// TIA Portal V20 export
DATA_BLOCK "Config"   // DB45
{ DB_Accessible_From_OPC_UA := 'FALSE' }
AUTHOR : ERsystem_FA2_DH. Kim
// stored: Access Published, DBAccessibleFromOPCUA false, DBAccessibleFromWebserver false, MemoryReserve 100, Namespace Unit1.Em7
   VAR RETAIN
      em { ExternalAccessible := 'False'; ExternalVisible := 'False'; ExternalWritable := 'False'} : "LAF_typeEmConfiguration";
      axis { ExternalAccessible := 'False'; ExternalVisible := 'False'; ExternalWritable := 'False'} : Array[1.._.U1EM7_NO_OF_AXES] of DB_ANY;
      cam { ExternalAccessible := 'False'; ExternalVisible := 'False'; ExternalWritable := 'False'} : Array[1.._.U1EM7_NO_OF_CAM] of DB_ANY;
      cmSepaClampDetectSensor { ExternalAccessible := 'False'; ExternalVisible := 'False'; ExternalWritable := 'False'} : "LBC_typeDigitalSignalConfiguration";
      cmSepaGripperDetectSensor { ExternalAccessible := 'False'; ExternalVisible := 'False'; ExternalWritable := 'False'} : "LBC_typeDigitalSignalConfiguration";
      cmJRWinderDetectSensor { ExternalAccessible := 'False'; ExternalVisible := 'False'; ExternalWritable := 'False'} : "LBC_typeDigitalSignalConfiguration";
      cmSepaClampSafetyPinDetectSensor { ExternalAccessible := 'False'; ExternalVisible := 'False'; ExternalWritable := 'False'} : "LBC_typeDigitalSignalConfiguration";
      cmSepaGripperSafetyPinDetectSensor { ExternalAccessible := 'False'; ExternalVisible := 'False'; ExternalWritable := 'False'} : "LBC_typeDigitalSignalConfiguration";
      cmSepaClampnCutterAxisX { ExternalAccessible := 'False'; ExternalVisible := 'False'; ExternalWritable := 'False'} : "LBC_typeAxis64PosConfiguration";
      cmSepaClampnCutterAxisZ { ExternalAccessible := 'False'; ExternalVisible := 'False'; ExternalWritable := 'False'} : "LBC_typeAxis64PosConfiguration";
      cmSepaGripperAxisX { ExternalAccessible := 'False'; ExternalVisible := 'False'; ExternalWritable := 'False'} : "LBC_typeAxis64PosConfiguration";
      cmSepaGripperAxisZ { ExternalAccessible := 'False'; ExternalVisible := 'False'; ExternalWritable := 'False'} : "LBC_typeAxis64PosConfiguration";
      cmSepaGripperAxisC { ExternalAccessible := 'False'; ExternalVisible := 'False'; ExternalWritable := 'False'} : "LBC_typeAxis64PosConfiguration";
      cmJRWinderRearAxisY { ExternalAccessible := 'False'; ExternalVisible := 'False'; ExternalWritable := 'False'} : "LBC_typeAxis64PosConfiguration";
      cmJRWinderFrontAxisY { ExternalAccessible := 'False'; ExternalVisible := 'False'; ExternalWritable := 'False'} : "LBC_typeAxis64PosConfiguration";
      cmJRWinderAxisB { ExternalAccessible := 'False'; ExternalVisible := 'False'; ExternalWritable := 'False'} : "LBC_typeAxis64PosConfiguration";
      cmJRPusherAxisZ { ExternalAccessible := 'False'; ExternalVisible := 'False'; ExternalWritable := 'False'} : "LBC_typeAxis64PosConfiguration";
      cmSepaCutterUpDown { ExternalAccessible := 'False'; ExternalVisible := 'False'; ExternalWritable := 'False'} : "LBC_typeTwoWayActuatorConfiguration";
      cmSepaClampTopUpDown { ExternalAccessible := 'False'; ExternalVisible := 'False'; ExternalWritable := 'False'} : "LBC_typeTwoWayActuatorConfiguration";
      cmSepaClampBottomUpDown { ExternalAccessible := 'False'; ExternalVisible := 'False'; ExternalWritable := 'False'} : "LBC_typeTwoWayActuatorConfiguration";
      cmStackGripperOpenClose { ExternalAccessible := 'False'; ExternalVisible := 'False'; ExternalWritable := 'False'} : "LBC_typeTwoWayActuatorConfiguration";
      cmStackGripperFwdBwd { ExternalAccessible := 'False'; ExternalVisible := 'False'; ExternalWritable := 'False'} : "LBC_typeTwoWayActuatorConfiguration";
      cmJRWinderClampTopRearUpDown { ExternalAccessible := 'False'; ExternalVisible := 'False'; ExternalWritable := 'False'} : "LBC_typeTwoWayActuatorConfiguration";
      cmJRWinderClampBtmRearUpDown { ExternalAccessible := 'False'; ExternalVisible := 'False'; ExternalWritable := 'False'} : "LBC_typeTwoWayActuatorConfiguration";
      cmJRWinderClampTopFrontUpDown { ExternalAccessible := 'False'; ExternalVisible := 'False'; ExternalWritable := 'False'} : "LBC_typeTwoWayActuatorConfiguration";
      cmJRWinderClampBtmFrontUpDown { ExternalAccessible := 'False'; ExternalVisible := 'False'; ExternalWritable := 'False'} : "LBC_typeTwoWayActuatorConfiguration";
      cmPusherRollerUpDown { ExternalAccessible := 'False'; ExternalVisible := 'False'; ExternalWritable := 'False'} : "LBC_typeTwoWayActuatorConfiguration";
      cmPusherRollerFwdBwd { ExternalAccessible := 'False'; ExternalVisible := 'False'; ExternalWritable := 'False'} : "LBC_typeTwoWayActuatorConfiguration";
      softCam : Struct
         cmSepaClampnCutterAxisX : "LER_typeSoftCamInterface";
         cmSepaClampnCutterAxisZ { S7_SetPoint := 'True'} : "LER_typeSoftCamInterface";
         cmSepaGripperAxisX { S7_SetPoint := 'True'} : "LER_typeSoftCamInterface";
         cmSepaGripperAxisZ { S7_SetPoint := 'True'} : "LER_typeSoftCamInterface";
         cmSepaGripperAxisC { S7_SetPoint := 'True'} : "LER_typeSoftCamInterface";
         cmJRWinderRearAxisY { S7_SetPoint := 'True'} : "LER_typeSoftCamInterface";
         cmJRWinderFrontAxisY { S7_SetPoint := 'True'} : "LER_typeSoftCamInterface";
         cmJRWinderAxisB { S7_SetPoint := 'True'} : "LER_typeSoftCamInterface";
         cmJRPusherAxisZ { S7_SetPoint := 'True'} : "LER_typeSoftCamInterface";
      END_STRUCT;
   END_VAR
BEGIN
   em.referenceDesignator.parent := WSTRING#'';
   em.referenceDesignator.relative := WSTRING#'';
   em.referenceDesignator.combined := WSTRING#'';
   axis[1] := 177;   // SepaClampnCutterAxisX
   axis[2] := 175;   // SepaClampnCutterAxisZ
   axis[3] := 178;   // SepaGripperAxisX
   axis[4] := 173;   // SepaGripperAxisZ
   axis[5] := 174;   // SepaGripperAxisC
   axis[6] := 180;   // JRWinderRearAxisY
   axis[7] := 179;   // JRWinderFrontAxisY
   axis[8] := 176;   // JRWinderAxisB
   axis[9] := 141;   // JRPusherAxisZ
   cam[1] := 184;
   cam[2] := 23;
   cam[3] := 266;
   cam[4] := 47;
   cam[5] := 390;
   cam[6] := 80;
   cmSepaClampDetectSensor.referenceDesignator := WSTRING#'DigitalSignal';
   cmSepaClampDetectSensor.onDelay := T#0MS;
   cmSepaClampDetectSensor.offDelay := T#0MS;
   cmSepaClampDetectSensor.default := FALSE;
   cmSepaClampDetectSensor.invertProcessValue := FALSE;
   cmSepaClampDetectSensor.disableAlarms := FALSE;
   cmSepaGripperDetectSensor.referenceDesignator := WSTRING#'DigitalSignal';
   cmSepaGripperDetectSensor.onDelay := T#0MS;
   cmSepaGripperDetectSensor.offDelay := T#0MS;
   cmSepaGripperDetectSensor.default := FALSE;
   cmSepaGripperDetectSensor.invertProcessValue := FALSE;
   cmSepaGripperDetectSensor.disableAlarms := FALSE;
   cmJRWinderDetectSensor.referenceDesignator := WSTRING#'DigitalSignal';
   cmJRWinderDetectSensor.onDelay := T#0MS;
   cmJRWinderDetectSensor.offDelay := T#0MS;
   cmJRWinderDetectSensor.default := FALSE;
   cmJRWinderDetectSensor.invertProcessValue := FALSE;
   cmJRWinderDetectSensor.disableAlarms := FALSE;
   cmSepaClampSafetyPinDetectSensor.referenceDesignator := WSTRING#'DigitalSignal';
   cmSepaClampSafetyPinDetectSensor.onDelay := T#0MS;
   cmSepaClampSafetyPinDetectSensor.offDelay := T#0MS;
   cmSepaClampSafetyPinDetectSensor.default := FALSE;
   cmSepaClampSafetyPinDetectSensor.invertProcessValue := FALSE;
   cmSepaClampSafetyPinDetectSensor.disableAlarms := FALSE;
   cmSepaGripperSafetyPinDetectSensor.referenceDesignator := WSTRING#'DigitalSignal';
   cmSepaGripperSafetyPinDetectSensor.onDelay := T#0MS;
   cmSepaGripperSafetyPinDetectSensor.offDelay := T#0MS;
   cmSepaGripperSafetyPinDetectSensor.default := FALSE;
   cmSepaGripperSafetyPinDetectSensor.invertProcessValue := FALSE;
   cmSepaGripperSafetyPinDetectSensor.disableAlarms := FALSE;
   cmSepaClampnCutterAxisX.referenceDesignator := WSTRING#'SepaClampnCutterAxisX';
   cmSepaClampnCutterAxisX.disableAlarms := FALSE;
   cmSepaClampnCutterAxisX.masterControlPopUp := TRUE;
   cmSepaClampnCutterAxisX.setPositions[0].position := 100.0;
   cmSepaClampnCutterAxisX.setPositions[1].position := 0.0;
   cmSepaClampnCutterAxisX.setPositions[2].position := 200.0;
   cmSepaClampnCutterAxisX.setPositions[3].position := 106.125;
   cmSepaClampnCutterAxisX.setPositions[4].position := 212.25;
   cmSepaClampnCutterAxisX.setPositions[5].position := 318.375;
   cmSepaClampnCutterAxisX.setPositions[6].position := 424.5;
   cmSepaClampnCutterAxisX.setPositions[7].position := 600.0;
   cmSepaClampnCutterAxisX.setPositions[8..15].position := 0.0;
   cmSepaClampnCutterAxisX.setPositions[0..2].velocity := 100.0;
   cmSepaClampnCutterAxisX.setPositions[3..6].velocity := -1.17916666666667;
   cmSepaClampnCutterAxisX.setPositions[7].velocity := 100.0;
   cmSepaClampnCutterAxisX.setPositions[8..15].velocity := -1.0;
   cmSepaClampnCutterAxisX.setPositions[0..2].acceleration := 1000.0;
   cmSepaClampnCutterAxisX.setPositions[3..6].acceleration := -11.7916666666667;
   cmSepaClampnCutterAxisX.setPositions[7].acceleration := 1000.0;
   cmSepaClampnCutterAxisX.setPositions[8..15].acceleration := -1.0;
   cmSepaClampnCutterAxisX.setPositions[0..2].deceleration := 1000.0;
   cmSepaClampnCutterAxisX.setPositions[3..6].deceleration := -11.7916666666667;
   cmSepaClampnCutterAxisX.setPositions[7].deceleration := 1000.0;
   cmSepaClampnCutterAxisX.setPositions[8..15].deceleration := -1.0;
   cmSepaClampnCutterAxisX.setPositions[0..15]."name" := '';
   cmSepaClampnCutterAxisZ.referenceDesignator := WSTRING#'SepaClampnCutterAxisZ';
   cmSepaClampnCutterAxisZ.disableAlarms := FALSE;
   cmSepaClampnCutterAxisZ.masterControlPopUp := TRUE;
   cmSepaClampnCutterAxisZ.setPositions[0].position := 0.0;
   cmSepaClampnCutterAxisZ.setPositions[1].position := 25.0;
   cmSepaClampnCutterAxisZ.setPositions[2].position := 50.0;
   cmSepaClampnCutterAxisZ.setPositions[3].position := -106.125;
   cmSepaClampnCutterAxisZ.setPositions[4..15].position := 0.0;
   cmSepaClampnCutterAxisZ.setPositions[0..2].velocity := 50.0;
   cmSepaClampnCutterAxisZ.setPositions[3..4].velocity := -1.17916666666667;
   cmSepaClampnCutterAxisZ.setPositions[5..15].velocity := -1.0;
   cmSepaClampnCutterAxisZ.setPositions[0..2].acceleration := 500.0;
   cmSepaClampnCutterAxisZ.setPositions[3..4].acceleration := -11.7916666666667;
   cmSepaClampnCutterAxisZ.setPositions[5..15].acceleration := -1.0;
   cmSepaClampnCutterAxisZ.setPositions[0..2].deceleration := 500.0;
   cmSepaClampnCutterAxisZ.setPositions[3..4].deceleration := -11.7916666666667;
   cmSepaClampnCutterAxisZ.setPositions[5..15].deceleration := -1.0;
   cmSepaClampnCutterAxisZ.setPositions[0..15]."name" := '';
   cmSepaGripperAxisX.referenceDesignator := WSTRING#'SepaGripperAxisX';
   cmSepaGripperAxisX.disableAlarms := FALSE;
   cmSepaGripperAxisX.masterControlPopUp := TRUE;
   cmSepaGripperAxisX.setPositions[0].position := 100.0;
   cmSepaGripperAxisX.setPositions[1].position := 400.0;
   cmSepaGripperAxisX.setPositions[2].position := 300.0;
   cmSepaGripperAxisX.setPositions[3].position := 150.0;
   cmSepaGripperAxisX.setPositions[4].position := 250.0;
   cmSepaGripperAxisX.setPositions[5].position := 100.0;
   cmSepaGripperAxisX.setPositions[6..15].position := 0.0;
   cmSepaGripperAxisX.setPositions[0..6].velocity := 100.0;
   cmSepaGripperAxisX.setPositions[7..15].velocity := -1.0;
   cmSepaGripperAxisX.setPositions[0..6].acceleration := 1000.0;
   cmSepaGripperAxisX.setPositions[7..15].acceleration := -1.0;
   cmSepaGripperAxisX.setPositions[0..6].deceleration := 1000.0;
   cmSepaGripperAxisX.setPositions[7..15].deceleration := -1.0;
   cmSepaGripperAxisX.setPositions[0..15]."name" := '';
   cmSepaGripperAxisZ.referenceDesignator := WSTRING#'SepaGripperAxisZ';
   cmSepaGripperAxisZ.disableAlarms := FALSE;
   cmSepaGripperAxisZ.masterControlPopUp := TRUE;
   cmSepaGripperAxisZ.setPositions[0].position := 0.0;
   cmSepaGripperAxisZ.setPositions[1].position := 25.0;
   cmSepaGripperAxisZ.setPositions[2].position := 2.0;
   cmSepaGripperAxisZ.setPositions[3].position := 3.0;
   cmSepaGripperAxisZ.setPositions[4].position := 4.0;
   cmSepaGripperAxisZ.setPositions[5].position := 5.0;
   cmSepaGripperAxisZ.setPositions[6].position := 50.0;
   cmSepaGripperAxisZ.setPositions[7..15].position := 0.0;
   cmSepaGripperAxisZ.setPositions[0..6].velocity := 50.0;
   cmSepaGripperAxisZ.setPositions[7..15].velocity := -1.0;
   cmSepaGripperAxisZ.setPositions[0..6].acceleration := 500.0;
   cmSepaGripperAxisZ.setPositions[7..15].acceleration := -1.0;
   cmSepaGripperAxisZ.setPositions[0..6].deceleration := 500.0;
   cmSepaGripperAxisZ.setPositions[7..15].deceleration := -1.0;
   cmSepaGripperAxisZ.setPositions[0..15]."name" := '';
   cmSepaGripperAxisC.referenceDesignator := WSTRING#'SepaGripperAxisC';
   cmSepaGripperAxisC.disableAlarms := FALSE;
   cmSepaGripperAxisC.masterControlPopUp := TRUE;
   cmSepaGripperAxisC.setPositions[0].position := 0.0;
   cmSepaGripperAxisC.setPositions[1].position := 180.0;
   cmSepaGripperAxisC.setPositions[2].position := 90.0;
   cmSepaGripperAxisC.setPositions[3..15].position := 0.0;
   cmSepaGripperAxisC.setPositions[0..2].velocity := 100.0;
   cmSepaGripperAxisC.setPositions[3..15].velocity := -1.0;
   cmSepaGripperAxisC.setPositions[0..2].acceleration := 1000.0;
   cmSepaGripperAxisC.setPositions[3..15].acceleration := -1.0;
   cmSepaGripperAxisC.setPositions[0..2].deceleration := 1000.0;
   cmSepaGripperAxisC.setPositions[3..15].deceleration := -1.0;
   cmSepaGripperAxisC.setPositions[0..15]."name" := '';
   cmJRWinderRearAxisY.referenceDesignator := WSTRING#'JRWinderRearAxisY';
   cmJRWinderRearAxisY.disableAlarms := FALSE;
   cmJRWinderRearAxisY.masterControlPopUp := TRUE;
   cmJRWinderRearAxisY.setPositions[0].position := 0.0;
   cmJRWinderRearAxisY.setPositions[1].position := 50.0;
   cmJRWinderRearAxisY.setPositions[2..15].position := 0.0;
   cmJRWinderRearAxisY.setPositions[0..1].velocity := 50.0;
   cmJRWinderRearAxisY.setPositions[2..15].velocity := -1.0;
   cmJRWinderRearAxisY.setPositions[0..1].acceleration := 500.0;
   cmJRWinderRearAxisY.setPositions[2..15].acceleration := -1.0;
   cmJRWinderRearAxisY.setPositions[0..1].deceleration := 500.0;
   cmJRWinderRearAxisY.setPositions[2..15].deceleration := -1.0;
   cmJRWinderRearAxisY.setPositions[0..15]."name" := '';
   cmJRWinderFrontAxisY.referenceDesignator := WSTRING#'JRWinderFrontAxisY';
   cmJRWinderFrontAxisY.disableAlarms := FALSE;
   cmJRWinderFrontAxisY.masterControlPopUp := TRUE;
   cmJRWinderFrontAxisY.setPositions[0].position := 0.0;
   cmJRWinderFrontAxisY.setPositions[1].position := 50.0;
   cmJRWinderFrontAxisY.setPositions[2..15].position := 0.0;
   cmJRWinderFrontAxisY.setPositions[0..1].velocity := 50.0;
   cmJRWinderFrontAxisY.setPositions[2..15].velocity := -1.0;
   cmJRWinderFrontAxisY.setPositions[0..1].acceleration := 500.0;
   cmJRWinderFrontAxisY.setPositions[2..15].acceleration := -1.0;
   cmJRWinderFrontAxisY.setPositions[0..1].deceleration := 500.0;
   cmJRWinderFrontAxisY.setPositions[2..15].deceleration := -1.0;
   cmJRWinderFrontAxisY.setPositions[0..15]."name" := '';
   cmJRWinderAxisB.referenceDesignator := WSTRING#'JRWinderAxisB';
   cmJRWinderAxisB.disableAlarms := FALSE;
   cmJRWinderAxisB.masterControlPopUp := TRUE;
   cmJRWinderAxisB.setPositions[0].position := 0.0;
   cmJRWinderAxisB.setPositions[1].position := 90.0;
   cmJRWinderAxisB.setPositions[2].position := 180.0;
   cmJRWinderAxisB.setPositions[3].position := 270.0;
   cmJRWinderAxisB.setPositions[4].position := 360.0;
   cmJRWinderAxisB.setPositions[5].position := 450.0;
   cmJRWinderAxisB.setPositions[6].position := 540.0;
   cmJRWinderAxisB.setPositions[7].position := 360.0;
   cmJRWinderAxisB.setPositions[8].position := 540.0;
   cmJRWinderAxisB.setPositions[9..15].position := 0.0;
   cmJRWinderAxisB.setPositions[0..8].velocity := 100.0;
   cmJRWinderAxisB.setPositions[9..15].velocity := -1.0;
   cmJRWinderAxisB.setPositions[0..8].acceleration := 1000.0;
   cmJRWinderAxisB.setPositions[9..15].acceleration := -1.0;
   cmJRWinderAxisB.setPositions[0..8].deceleration := 1000.0;
   cmJRWinderAxisB.setPositions[9..15].deceleration := -1.0;
   cmJRWinderAxisB.setPositions[0..15]."name" := '';
   cmJRPusherAxisZ.referenceDesignator := WSTRING#'JRPusherAxisZ';
   cmJRPusherAxisZ.disableAlarms := FALSE;
   cmJRPusherAxisZ.masterControlPopUp := TRUE;
   cmJRPusherAxisZ.setPositions[0].position := 0.0;
   cmJRPusherAxisZ.setPositions[1].position := 100.0;
   cmJRPusherAxisZ.setPositions[2].position := -106.125;
   cmJRPusherAxisZ.setPositions[3..15].position := 0.0;
   cmJRPusherAxisZ.setPositions[0..1].velocity := 100.0;
   cmJRPusherAxisZ.setPositions[2..3].velocity := -1.17916666666667;
   cmJRPusherAxisZ.setPositions[4..15].velocity := -1.0;
   cmJRPusherAxisZ.setPositions[0..1].acceleration := 1000.0;
   cmJRPusherAxisZ.setPositions[2..3].acceleration := -11.7916666666667;
   cmJRPusherAxisZ.setPositions[4..15].acceleration := -1.0;
   cmJRPusherAxisZ.setPositions[0..1].deceleration := 1000.0;
   cmJRPusherAxisZ.setPositions[2..3].deceleration := -11.7916666666667;
   cmJRPusherAxisZ.setPositions[4..15].deceleration := -1.0;
   cmJRPusherAxisZ.setPositions[0..15]."name" := '';
   cmSepaCutterUpDown.referenceDesignator := WSTRING#'SepaCutterUpDown';
   cmSepaCutterUpDown.monitoringLeavingFeedback := T#5S;
   cmSepaCutterUpDown.monitoringReachingFeedback := T#5S;
   cmSepaCutterUpDown.monitoringDiscrepancy := T#0MS;
   cmSepaCutterUpDown.setOutputHomeContinuously := TRUE;
   cmSepaCutterUpDown.setOutputWorkContinuously := TRUE;
   cmSepaCutterUpDown.disableHomeCommand := FALSE;
   cmSepaCutterUpDown.disableFeedbackHomePos := FALSE;
   cmSepaCutterUpDown.disableFeedbackWorkPos := FALSE;
   cmSepaCutterUpDown.disableAlarms := FALSE;
   cmSepaCutterUpDown.resetOutputsOnError := FALSE;
   cmSepaCutterUpDown.allwaysWaitOnReachingTime := FALSE;
   cmSepaClampTopUpDown.referenceDesignator := WSTRING#'SepaClampTopUpDown';
   cmSepaClampTopUpDown.monitoringLeavingFeedback := T#5S;
   cmSepaClampTopUpDown.monitoringReachingFeedback := T#5S;
   cmSepaClampTopUpDown.monitoringDiscrepancy := T#0MS;
   cmSepaClampTopUpDown.setOutputHomeContinuously := TRUE;
   cmSepaClampTopUpDown.setOutputWorkContinuously := TRUE;
   cmSepaClampTopUpDown.disableHomeCommand := FALSE;
   cmSepaClampTopUpDown.disableFeedbackHomePos := FALSE;
   cmSepaClampTopUpDown.disableFeedbackWorkPos := FALSE;
   cmSepaClampTopUpDown.disableAlarms := FALSE;
   cmSepaClampTopUpDown.resetOutputsOnError := FALSE;
   cmSepaClampTopUpDown.allwaysWaitOnReachingTime := FALSE;
   cmSepaClampBottomUpDown.referenceDesignator := WSTRING#'ClampBottomUpDown';
   cmSepaClampBottomUpDown.monitoringLeavingFeedback := T#5S;
   cmSepaClampBottomUpDown.monitoringReachingFeedback := T#5S;
   cmSepaClampBottomUpDown.monitoringDiscrepancy := T#0MS;
   cmSepaClampBottomUpDown.setOutputHomeContinuously := TRUE;
   cmSepaClampBottomUpDown.setOutputWorkContinuously := TRUE;
   cmSepaClampBottomUpDown.disableHomeCommand := FALSE;
   cmSepaClampBottomUpDown.disableFeedbackHomePos := FALSE;
   cmSepaClampBottomUpDown.disableFeedbackWorkPos := FALSE;
   cmSepaClampBottomUpDown.disableAlarms := FALSE;
   cmSepaClampBottomUpDown.resetOutputsOnError := FALSE;
   cmSepaClampBottomUpDown.allwaysWaitOnReachingTime := FALSE;
   cmStackGripperOpenClose.referenceDesignator := WSTRING#'GripperOpenClose';
   cmStackGripperOpenClose.monitoringLeavingFeedback := T#1S;
   cmStackGripperOpenClose.monitoringReachingFeedback := T#1S;
   cmStackGripperOpenClose.monitoringDiscrepancy := T#0MS;
   cmStackGripperOpenClose.setOutputHomeContinuously := TRUE;
   cmStackGripperOpenClose.setOutputWorkContinuously := TRUE;
   cmStackGripperOpenClose.disableHomeCommand := FALSE;
   cmStackGripperOpenClose.disableFeedbackHomePos := FALSE;
   cmStackGripperOpenClose.disableFeedbackWorkPos := FALSE;
   cmStackGripperOpenClose.disableAlarms := FALSE;
   cmStackGripperOpenClose.resetOutputsOnError := FALSE;
   cmStackGripperOpenClose.allwaysWaitOnReachingTime := FALSE;
   cmStackGripperFwdBwd.referenceDesignator := WSTRING#'GripperFwdBwd';
   cmStackGripperFwdBwd.monitoringLeavingFeedback := T#1S;
   cmStackGripperFwdBwd.monitoringReachingFeedback := T#1S;
   cmStackGripperFwdBwd.monitoringDiscrepancy := T#0MS;
   cmStackGripperFwdBwd.setOutputHomeContinuously := TRUE;
   cmStackGripperFwdBwd.setOutputWorkContinuously := TRUE;
   cmStackGripperFwdBwd.disableHomeCommand := FALSE;
   cmStackGripperFwdBwd.disableFeedbackHomePos := FALSE;
   cmStackGripperFwdBwd.disableFeedbackWorkPos := FALSE;
   cmStackGripperFwdBwd.disableAlarms := FALSE;
   cmStackGripperFwdBwd.resetOutputsOnError := FALSE;
   cmStackGripperFwdBwd.allwaysWaitOnReachingTime := FALSE;
   cmJRWinderClampTopRearUpDown.referenceDesignator := WSTRING#'JRClampTopRearUpDown.';
   cmJRWinderClampTopRearUpDown.monitoringLeavingFeedback := T#1S;
   cmJRWinderClampTopRearUpDown.monitoringReachingFeedback := T#1S;
   cmJRWinderClampTopRearUpDown.monitoringDiscrepancy := T#0MS;
   cmJRWinderClampTopRearUpDown.setOutputHomeContinuously := TRUE;
   cmJRWinderClampTopRearUpDown.setOutputWorkContinuously := TRUE;
   cmJRWinderClampTopRearUpDown.disableHomeCommand := FALSE;
   cmJRWinderClampTopRearUpDown.disableFeedbackHomePos := TRUE;
   cmJRWinderClampTopRearUpDown.disableFeedbackWorkPos := TRUE;
   cmJRWinderClampTopRearUpDown.disableAlarms := FALSE;
   cmJRWinderClampTopRearUpDown.resetOutputsOnError := FALSE;
   cmJRWinderClampTopRearUpDown.allwaysWaitOnReachingTime := FALSE;
   cmJRWinderClampBtmRearUpDown.referenceDesignator := WSTRING#'JRClampBtmRearUpDown.';
   cmJRWinderClampBtmRearUpDown.monitoringLeavingFeedback := T#1S;
   cmJRWinderClampBtmRearUpDown.monitoringReachingFeedback := T#1S;
   cmJRWinderClampBtmRearUpDown.monitoringDiscrepancy := T#0MS;
   cmJRWinderClampBtmRearUpDown.setOutputHomeContinuously := TRUE;
   cmJRWinderClampBtmRearUpDown.setOutputWorkContinuously := TRUE;
   cmJRWinderClampBtmRearUpDown.disableHomeCommand := FALSE;
   cmJRWinderClampBtmRearUpDown.disableFeedbackHomePos := TRUE;
   cmJRWinderClampBtmRearUpDown.disableFeedbackWorkPos := TRUE;
   cmJRWinderClampBtmRearUpDown.disableAlarms := FALSE;
   cmJRWinderClampBtmRearUpDown.resetOutputsOnError := FALSE;
   cmJRWinderClampBtmRearUpDown.allwaysWaitOnReachingTime := FALSE;
   cmJRWinderClampTopFrontUpDown.referenceDesignator := WSTRING#'JRClampTopFrontUpDown.';
   cmJRWinderClampTopFrontUpDown.monitoringLeavingFeedback := T#1S;
   cmJRWinderClampTopFrontUpDown.monitoringReachingFeedback := T#1S;
   cmJRWinderClampTopFrontUpDown.monitoringDiscrepancy := T#0MS;
   cmJRWinderClampTopFrontUpDown.setOutputHomeContinuously := TRUE;
   cmJRWinderClampTopFrontUpDown.setOutputWorkContinuously := TRUE;
   cmJRWinderClampTopFrontUpDown.disableHomeCommand := FALSE;
   cmJRWinderClampTopFrontUpDown.disableFeedbackHomePos := TRUE;
   cmJRWinderClampTopFrontUpDown.disableFeedbackWorkPos := TRUE;
   cmJRWinderClampTopFrontUpDown.disableAlarms := FALSE;
   cmJRWinderClampTopFrontUpDown.resetOutputsOnError := FALSE;
   cmJRWinderClampTopFrontUpDown.allwaysWaitOnReachingTime := FALSE;
   cmJRWinderClampBtmFrontUpDown.referenceDesignator := WSTRING#'JRClampBtmFrontUpDown.';
   cmJRWinderClampBtmFrontUpDown.monitoringLeavingFeedback := T#1S;
   cmJRWinderClampBtmFrontUpDown.monitoringReachingFeedback := T#1S;
   cmJRWinderClampBtmFrontUpDown.monitoringDiscrepancy := T#0MS;
   cmJRWinderClampBtmFrontUpDown.setOutputHomeContinuously := TRUE;
   cmJRWinderClampBtmFrontUpDown.setOutputWorkContinuously := TRUE;
   cmJRWinderClampBtmFrontUpDown.disableHomeCommand := FALSE;
   cmJRWinderClampBtmFrontUpDown.disableFeedbackHomePos := TRUE;
   cmJRWinderClampBtmFrontUpDown.disableFeedbackWorkPos := TRUE;
   cmJRWinderClampBtmFrontUpDown.disableAlarms := FALSE;
   cmJRWinderClampBtmFrontUpDown.resetOutputsOnError := FALSE;
   cmJRWinderClampBtmFrontUpDown.allwaysWaitOnReachingTime := FALSE;
   cmPusherRollerUpDown.referenceDesignator := WSTRING#'PusherRollerUpDown';
   cmPusherRollerUpDown.monitoringLeavingFeedback := T#5S;
   cmPusherRollerUpDown.monitoringReachingFeedback := T#5S;
   cmPusherRollerUpDown.monitoringDiscrepancy := T#0MS;
   cmPusherRollerUpDown.setOutputHomeContinuously := TRUE;
   cmPusherRollerUpDown.setOutputWorkContinuously := TRUE;
   cmPusherRollerUpDown.disableHomeCommand := FALSE;
   cmPusherRollerUpDown.disableFeedbackHomePos := FALSE;
   cmPusherRollerUpDown.disableFeedbackWorkPos := FALSE;
   cmPusherRollerUpDown.disableAlarms := FALSE;
   cmPusherRollerUpDown.resetOutputsOnError := FALSE;
   cmPusherRollerUpDown.allwaysWaitOnReachingTime := FALSE;
   cmPusherRollerFwdBwd.referenceDesignator := WSTRING#'PusherRollerFwdBwd';
   cmPusherRollerFwdBwd.monitoringLeavingFeedback := T#5S;
   cmPusherRollerFwdBwd.monitoringReachingFeedback := T#5S;
   cmPusherRollerFwdBwd.monitoringDiscrepancy := T#0MS;
   cmPusherRollerFwdBwd.setOutputHomeContinuously := TRUE;
   cmPusherRollerFwdBwd.setOutputWorkContinuously := TRUE;
   cmPusherRollerFwdBwd.disableHomeCommand := FALSE;
   cmPusherRollerFwdBwd.disableFeedbackHomePos := FALSE;
   cmPusherRollerFwdBwd.disableFeedbackWorkPos := FALSE;
   cmPusherRollerFwdBwd.disableAlarms := FALSE;
   cmPusherRollerFwdBwd.resetOutputsOnError := FALSE;
   cmPusherRollerFwdBwd.allwaysWaitOnReachingTime := FALSE;
   softCam.cmSepaClampnCutterAxisX.TargetPosition := 0.0;
   softCam.cmSepaClampnCutterAxisX.ActualPosition := 0.0;
   softCam.cmSepaClampnCutterAxisX.UnitName := WSTRING#'';
   softCam.cmSepaClampnCutterAxisX.error := FALSE;
   softCam.cmSepaClampnCutterAxisX.status := 16#0000;
   softCam.cmSepaClampnCutterAxisX.position[0..15].SetValue.Negative := 0.0;
   softCam.cmSepaClampnCutterAxisX.position[0..15].SetValue.Postive := 0.0;
   softCam.cmSepaClampnCutterAxisX.position[0..15].ProcessValue.Postive := 0.0;
   softCam.cmSepaClampnCutterAxisX.position[0..15].ProcessValue.Negative := 0.0;
   softCam.cmSepaClampnCutterAxisX.position[0..15].ProcessValue.SetPos := 0.0;
   softCam.cmSepaClampnCutterAxisX.position[0..15].ProcessValue.inPos := FALSE;
   softCam.cmSepaClampnCutterAxisX.position[0..15].ProcessValue.isBefore := FALSE;
   softCam.cmSepaClampnCutterAxisX.position[0..15].ProcessValue.isAfter := FALSE;
   softCam.cmSepaClampnCutterAxisX.position[0..15].ProcessValue.PosName := WSTRING#'';
   softCam.cmSepaClampnCutterAxisZ.TargetPosition := 0.0;
   softCam.cmSepaClampnCutterAxisZ.ActualPosition := 0.0;
   softCam.cmSepaClampnCutterAxisZ.UnitName := WSTRING#'';
   softCam.cmSepaClampnCutterAxisZ.error := FALSE;
   softCam.cmSepaClampnCutterAxisZ.status := 16#0000;
   softCam.cmSepaClampnCutterAxisZ.position[0..15].SetValue.Negative := 0.0;
   softCam.cmSepaClampnCutterAxisZ.position[0..15].SetValue.Postive := 0.0;
   softCam.cmSepaClampnCutterAxisZ.position[0..15].ProcessValue.Postive := 0.0;
   softCam.cmSepaClampnCutterAxisZ.position[0..15].ProcessValue.Negative := 0.0;
   softCam.cmSepaClampnCutterAxisZ.position[0..15].ProcessValue.SetPos := 0.0;
   softCam.cmSepaClampnCutterAxisZ.position[0..15].ProcessValue.inPos := FALSE;
   softCam.cmSepaClampnCutterAxisZ.position[0..15].ProcessValue.isBefore := FALSE;
   softCam.cmSepaClampnCutterAxisZ.position[0..15].ProcessValue.isAfter := FALSE;
   softCam.cmSepaClampnCutterAxisZ.position[0..15].ProcessValue.PosName := WSTRING#'';
   softCam.cmSepaGripperAxisX.TargetPosition := 0.0;
   softCam.cmSepaGripperAxisX.ActualPosition := 0.0;
   softCam.cmSepaGripperAxisX.UnitName := WSTRING#'';
   softCam.cmSepaGripperAxisX.error := FALSE;
   softCam.cmSepaGripperAxisX.status := 16#0000;
   softCam.cmSepaGripperAxisX.position[0..15].SetValue.Negative := 0.0;
   softCam.cmSepaGripperAxisX.position[0..15].SetValue.Postive := 0.0;
   softCam.cmSepaGripperAxisX.position[0..15].ProcessValue.Postive := 0.0;
   softCam.cmSepaGripperAxisX.position[0..15].ProcessValue.Negative := 0.0;
   softCam.cmSepaGripperAxisX.position[0..15].ProcessValue.SetPos := 0.0;
   softCam.cmSepaGripperAxisX.position[0..15].ProcessValue.inPos := FALSE;
   softCam.cmSepaGripperAxisX.position[0..15].ProcessValue.isBefore := FALSE;
   softCam.cmSepaGripperAxisX.position[0..15].ProcessValue.isAfter := FALSE;
   softCam.cmSepaGripperAxisX.position[0..15].ProcessValue.PosName := WSTRING#'';
   softCam.cmSepaGripperAxisZ.TargetPosition := 0.0;
   softCam.cmSepaGripperAxisZ.ActualPosition := 0.0;
   softCam.cmSepaGripperAxisZ.UnitName := WSTRING#'';
   softCam.cmSepaGripperAxisZ.error := FALSE;
   softCam.cmSepaGripperAxisZ.status := 16#0000;
   softCam.cmSepaGripperAxisZ.position[0..15].SetValue.Negative := 0.0;
   softCam.cmSepaGripperAxisZ.position[0..15].SetValue.Postive := 0.0;
   softCam.cmSepaGripperAxisZ.position[0..15].ProcessValue.Postive := 0.0;
   softCam.cmSepaGripperAxisZ.position[0..15].ProcessValue.Negative := 0.0;
   softCam.cmSepaGripperAxisZ.position[0..15].ProcessValue.SetPos := 0.0;
   softCam.cmSepaGripperAxisZ.position[0..15].ProcessValue.inPos := FALSE;
   softCam.cmSepaGripperAxisZ.position[0..15].ProcessValue.isBefore := FALSE;
   softCam.cmSepaGripperAxisZ.position[0..15].ProcessValue.isAfter := FALSE;
   softCam.cmSepaGripperAxisZ.position[0..15].ProcessValue.PosName := WSTRING#'';
   softCam.cmSepaGripperAxisC.TargetPosition := 0.0;
   softCam.cmSepaGripperAxisC.ActualPosition := 0.0;
   softCam.cmSepaGripperAxisC.UnitName := WSTRING#'';
   softCam.cmSepaGripperAxisC.error := FALSE;
   softCam.cmSepaGripperAxisC.status := 16#0000;
   softCam.cmSepaGripperAxisC.position[0..15].SetValue.Negative := 0.0;
   softCam.cmSepaGripperAxisC.position[0..15].SetValue.Postive := 0.0;
   softCam.cmSepaGripperAxisC.position[0..15].ProcessValue.Postive := 0.0;
   softCam.cmSepaGripperAxisC.position[0..15].ProcessValue.Negative := 0.0;
   softCam.cmSepaGripperAxisC.position[0..15].ProcessValue.SetPos := 0.0;
   softCam.cmSepaGripperAxisC.position[0..15].ProcessValue.inPos := FALSE;
   softCam.cmSepaGripperAxisC.position[0..15].ProcessValue.isBefore := FALSE;
   softCam.cmSepaGripperAxisC.position[0..15].ProcessValue.isAfter := FALSE;
   softCam.cmSepaGripperAxisC.position[0..15].ProcessValue.PosName := WSTRING#'';
   softCam.cmJRWinderRearAxisY.TargetPosition := 0.0;
   softCam.cmJRWinderRearAxisY.ActualPosition := 0.0;
   softCam.cmJRWinderRearAxisY.UnitName := WSTRING#'';
   softCam.cmJRWinderRearAxisY.error := FALSE;
   softCam.cmJRWinderRearAxisY.status := 16#0000;
   softCam.cmJRWinderRearAxisY.position[0..15].SetValue.Negative := 0.0;
   softCam.cmJRWinderRearAxisY.position[0..15].SetValue.Postive := 0.0;
   softCam.cmJRWinderRearAxisY.position[0..15].ProcessValue.Postive := 0.0;
   softCam.cmJRWinderRearAxisY.position[0..15].ProcessValue.Negative := 0.0;
   softCam.cmJRWinderRearAxisY.position[0..15].ProcessValue.SetPos := 0.0;
   softCam.cmJRWinderRearAxisY.position[0..15].ProcessValue.inPos := FALSE;
   softCam.cmJRWinderRearAxisY.position[0..15].ProcessValue.isBefore := FALSE;
   softCam.cmJRWinderRearAxisY.position[0..15].ProcessValue.isAfter := FALSE;
   softCam.cmJRWinderRearAxisY.position[0..15].ProcessValue.PosName := WSTRING#'';
   softCam.cmJRWinderFrontAxisY.TargetPosition := 0.0;
   softCam.cmJRWinderFrontAxisY.ActualPosition := 0.0;
   softCam.cmJRWinderFrontAxisY.UnitName := WSTRING#'';
   softCam.cmJRWinderFrontAxisY.error := FALSE;
   softCam.cmJRWinderFrontAxisY.status := 16#0000;
   softCam.cmJRWinderFrontAxisY.position[0..15].SetValue.Negative := 0.0;
   softCam.cmJRWinderFrontAxisY.position[0..15].SetValue.Postive := 0.0;
   softCam.cmJRWinderFrontAxisY.position[0..15].ProcessValue.Postive := 0.0;
   softCam.cmJRWinderFrontAxisY.position[0..15].ProcessValue.Negative := 0.0;
   softCam.cmJRWinderFrontAxisY.position[0..15].ProcessValue.SetPos := 0.0;
   softCam.cmJRWinderFrontAxisY.position[0..15].ProcessValue.inPos := FALSE;
   softCam.cmJRWinderFrontAxisY.position[0..15].ProcessValue.isBefore := FALSE;
   softCam.cmJRWinderFrontAxisY.position[0..15].ProcessValue.isAfter := FALSE;
   softCam.cmJRWinderFrontAxisY.position[0..15].ProcessValue.PosName := WSTRING#'';
   softCam.cmJRWinderAxisB.TargetPosition := 0.0;
   softCam.cmJRWinderAxisB.ActualPosition := 0.0;
   softCam.cmJRWinderAxisB.UnitName := WSTRING#'';
   softCam.cmJRWinderAxisB.error := FALSE;
   softCam.cmJRWinderAxisB.status := 16#0000;
   softCam.cmJRWinderAxisB.position[0..15].SetValue.Negative := 0.0;
   softCam.cmJRWinderAxisB.position[0..15].SetValue.Postive := 0.0;
   softCam.cmJRWinderAxisB.position[0..15].ProcessValue.Postive := 0.0;
   softCam.cmJRWinderAxisB.position[0..15].ProcessValue.Negative := 0.0;
   softCam.cmJRWinderAxisB.position[0..15].ProcessValue.SetPos := 0.0;
   softCam.cmJRWinderAxisB.position[0..15].ProcessValue.inPos := FALSE;
   softCam.cmJRWinderAxisB.position[0..15].ProcessValue.isBefore := FALSE;
   softCam.cmJRWinderAxisB.position[0..15].ProcessValue.isAfter := FALSE;
   softCam.cmJRWinderAxisB.position[0..15].ProcessValue.PosName := WSTRING#'';
   softCam.cmJRPusherAxisZ.TargetPosition := 0.0;
   softCam.cmJRPusherAxisZ.ActualPosition := 0.0;
   softCam.cmJRPusherAxisZ.UnitName := WSTRING#'';
   softCam.cmJRPusherAxisZ.error := FALSE;
   softCam.cmJRPusherAxisZ.status := 16#0000;
   softCam.cmJRPusherAxisZ.position[0..15].SetValue.Negative := 0.0;
   softCam.cmJRPusherAxisZ.position[0..15].SetValue.Postive := 0.0;
   softCam.cmJRPusherAxisZ.position[0..15].ProcessValue.Postive := 0.0;
   softCam.cmJRPusherAxisZ.position[0..15].ProcessValue.Negative := 0.0;
   softCam.cmJRPusherAxisZ.position[0..15].ProcessValue.SetPos := 0.0;
   softCam.cmJRPusherAxisZ.position[0..15].ProcessValue.inPos := FALSE;
   softCam.cmJRPusherAxisZ.position[0..15].ProcessValue.isBefore := FALSE;
   softCam.cmJRPusherAxisZ.position[0..15].ProcessValue.isAfter := FALSE;
   softCam.cmJRPusherAxisZ.position[0..15].ProcessValue.PosName := WSTRING#'';
END_DATA_BLOCK
